Staubli VAL3: D_ABZ_01.dtx

public aio aiEncCurrentPos = {link=e01CurrPos}
aio aiEncLatchedPos = {link=e01LatchPos}
aio aoEncResolution = {link=e01Counts}
aio aoPresetPos = {link=e01PrstPos}
public bool bLatchEnabled
bool bLatchLevel
bool bMemoLatchState
bool bPartLatched
bool bReset
dio diEncHwErr = {link=e01HwErr}
dio diEncLatched = {link=e01Latch}
dio diEncOvsErr = {link=e01OvsErr}
dio diLatchSignal = {link=e01LatchSig}
dio doEnableLatch = {link=e01EnLatch}
dio doEnablePreset = {link=e01EnPrst}
dio doLatchEdgFall = {link=e01LatchEdgFall}
dio doResetErr = {link=e01RstErr}
num nEncLatchedVal = 1
num nEncResolution = 1024
num nEncValue = 1
public num nLatchPeriod = 1
public num nMAXCOUNT
public num nMINCOUNT
num nPresetPos = 1
string sEncNum
string sTASK = "encoder"
